{attribute 'qualified_only'}
{attribute 'strict'}
{attribute 'to_string'}
TYPE E_KinStatus  :
(
    KinStatus_Error,            
    KinStatus_Empty,            
    KinStatus_Unknown,     
    KinStatus_StartPending, 
    KinStatus_Ready,         
    KinStatus_InvalidItfVersion := 16#4000
);
END_TYPE
//  KinStatus_InvalidItfVersion = '16#4000'

(* stored: Version 1.1.0.1
   EnumerationTextList E_KinStatus: Id {b8e75dbc-2280-42e0-abc0-b246ddd5ebd1} *)
